(* IEC 61131-3 sources: ArfBotOS/Codesys-4/ArfBotOS.fbsdev/Application.iecapp^/FUN/template/FB_PackML.fb.st^/wait, 6 files *)

(* ---- M_Aborted.meth.st ---- *)
METHOD PROTECTED M_Aborted : BOOL
VAR_INPUT
END_VAR

_SeqMain := 0;
_SeqAborting := 0;
_SeqClearing := 0;
_SeqCompleting := 0;
_SeqHolding := 0;
_SeqResetting := 0;
_SeqStarting := 0;
_SeqStopping := 0;
_SeqSuspending := 0;
_SeqUnholding := 0;
_SeqUnSuspending := 0;
END_METHOD

(* ---- M_Complete.meth.st ---- *)
METHOD PROTECTED M_Complete : BOOL
VAR_INPUT
END_VAR

(*_StateTimer.IN:=TRUE;

IF _StateTimer.Q THEN
	_StateTimer.IN:=FALSE;
	M_StateComplete();
END_IF*)
END_METHOD

(* ---- M_Held.meth.st ---- *)
METHOD PROTECTED M_Held : BOOL
VAR_INPUT
END_VAR

(*_StateTimer.IN:=TRUE;

IF _StateTimer.Q THEN
	_StateTimer.IN:=FALSE;
	M_StateComplete();
END_IF*)
END_METHOD

(* ---- M_Idle.meth.st ---- *)
METHOD PROTECTED M_Idle : BOOL
VAR_INPUT
END_VAR

(*_StateTimer.IN:=TRUE;

IF _StateTimer.Q THEN
	_StateTimer.IN:=FALSE;
	M_StateComplete();
END_IF*)
END_METHOD

(* ---- M_Stopped.meth.st ---- *)
METHOD PROTECTED M_Stopped : BOOL
VAR_INPUT
END_VAR

(*_StateTimer.IN:=TRUE;

IF _StateTimer.Q THEN
	_StateTimer.IN:=FALSE;
	M_StateComplete();
END_IF*)
END_METHOD

(* ---- M_Suspended.meth.st ---- *)
METHOD PROTECTED M_Suspended : BOOL
VAR_INPUT
END_VAR

(*_StateTimer.IN:=TRUE;

IF _StateTimer.Q THEN
	_StateTimer.IN:=FALSE;
	M_StateComplete();
END_IF*)
END_METHOD
